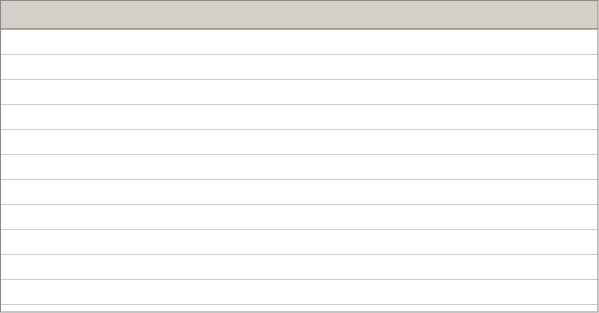
VISUALIZATION current  // 599x313
    Table (-1,-1 599x313), data array: AlarmManager.event_table_view.stAlarmEvents
        p3854506369: AlarmManager.event_table_view.stAlarmEvents[INDEX].nSourceId
        p1892666644: AlarmManager.event_table_view.stAlarmEvents[INDEX].nEventId
        p338671338: AlarmManager.event_table_view.stAlarmEvents[INDEX].Severity
        p2170511999: AlarmManager.event_table_view.stAlarmEvents[INDEX].ConfirmState
        p3723444502: AlarmManager.event_table_view.stAlarmEvents[INDEX].sDate
        p1218418051: AlarmManager.event_table_view.stAlarmEvents[INDEX].sTime
        p746581629: AlarmManager.event_table_view.stAlarmEvents[INDEX].Computer
        p3104783080: AlarmManager.event_table_view.stAlarmEvents[INDEX].sSource
        p2501879983: AlarmManager.event_table_view.stAlarmEvents[INDEX].MessageText
        p7306298: AlarmManager.event_table_view.stAlarmEvents[INDEX].bQuitMessage
        p1933151965: AlarmManager.event_table_view.stAlarmEvents[INDEX].bConfirmable
        p1755163831: 重要度
        p4092479075: 確認
        p2237128397: 日付
        p505689113: 時刻
        p2243050616: テキスト
        p1014161805: AlarmManager.event_table_view.DISP_ROWS - 1 + INT#1
END_VISUALIZATION

(* stored: Version 1.1.0.1
   Visu current: Id {2438d436-7f89-4bae-9c0b-71581f821792} *)
